Universal Robots PolyScope program: SandCube5.urp

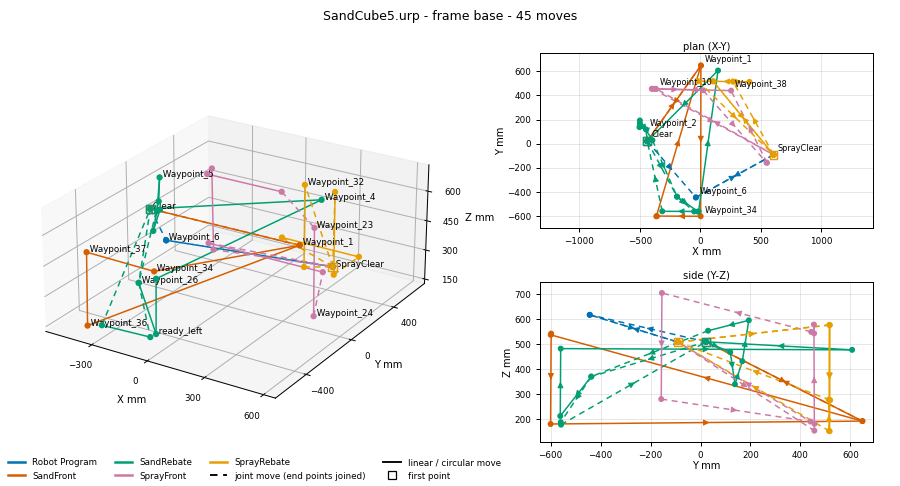
[picture p0: tool path of SandCube5.urp in frame base, 45 of 45 moves have a stored position in this frame; points joined in program order, loops and branches not executed]
Program SandCube5 (installation=sand5 directory=/programs createdIn=5.11.5.1010327 lastSavedIn=5.11.5.1010327 robotSerialNumber=20215500677)
Calibrated DH parameters: a=[0.000204, -0.239222, -0.391845, -0.000001, 0.000022, 0]; d=[0.162722, -355.808559, 353.37206, 2.570385, 0.099741, 0.099629]; alpha=[1.571124, 0.000988, 0.008295, 1.568963, -1.570303, 0]; deltaTheta=[0, -0.973091, 7.204745, 0.05153, 0, 0]
InitVariablesNode variables(variable(name=readyBackSand, expression=False), variable(name=readyFrontSand, expression=False), variable(name=readySpray, expression=False))
Robot Program (runOnlyOnce=false)
  Folder Main
    If readyFrontSand≟ True (checkContinuously=true)
      MoveJ speed 60 deg/s, acceleration 80 deg/s^2 (useActiveTCP=false positionType=JointAngles) tcp=DynabradeDual; feature=CubeFront
        Waypoint Clear: TCP in base x=-437.78 y=22.317 z=510.388 mm, rx=-1.2261 ry=-1.1914 rz=1.1915 rad; joints [-41.645, -103.017, 131.059, 99.527, -63.29, 31.09] deg; TCP offset x=3.18 y=114.64 z=98.2 mm, rx=-0.7854 ry=0 rz=0 rad; feature pose in base x=-591.611 y=-180.941 z=285.211 mm, rx=1.216 ry=1.1897 rz=1.1897 rad
        URCap Zero FT Sensor (Robotiq_Copilot, Robotiq Inc.) dataModel(NodeInitializedKey=true, WaitForSteadyWrenchOptionKey=true)
      Work := CubeFront
      Call SandFront
      Call SandRebate
      readyFrontSand := False
      Set DigitalOutput pin=digital_out[5]; digitalValue=0
    If readyBackSand≟ True (checkContinuously=true)
      Work := CubeFront
      Call SandFront
      readyBackSand := False
      Set DigitalOutput pin=digital_out[5]; digitalValue=0
    If readySpray≟ True (checkContinuously=true)
      MoveJ speed 60 deg/s, acceleration 80 deg/s^2 (useActiveTCP=false positionType=JointAngles) tcp=Spray; feature=SprayPlane
        Waypoint Waypoint_6: TCP in base x=-35.819 y=-443.732 z=618.465 mm, rx=1.57 ry=-0.053 rz=-0.0554 rad; joints [61.905, -86.892, 117.128, 101.277, -70.255, 21.732] deg; TCP offset x=20.839 y=-27.14 z=105.994 mm, rx=0.1226 ry=1.1769 rz=2.8697 rad; feature pose in base x=714.825 y=225.543 z=302.034 mm, rx=1.1969 ry=-1.2373 rz=-1.2135 rad
        Waypoint SprayClear: TCP in base x=607.137 y=-90.197 z=509.102 mm, rx=1.2034 ry=1.2067 rz=1.2159 rad; joints [154.541, -56.922, 94.352, -266.679, -69.476, 23.135] deg; TCP offset x=20.839 y=-27.14 z=105.994 mm, rx=0.1226 ry=1.1769 rz=2.8697 rad; feature pose in base x=807.673 y=110.818 z=310.566 mm, rx=1.2166 ry=-1.2106 rz=-1.2041 rad
        URCap Zero FT Sensor (Robotiq_Copilot, Robotiq Inc.) dataModel(NodeInitializedKey=true, WaitForSteadyWrenchOptionKey=true)
        Call SprayFront
        Call SprayRebate
        Waypoint Waypoint_6: TCP in base x=-35.819 y=-443.732 z=618.465 mm, rx=1.57 ry=-0.053 rz=-0.0554 rad; joints [61.905, -86.892, 117.128, 101.277, -70.255, 21.732] deg; TCP offset x=20.839 y=-27.14 z=105.994 mm, rx=0.1226 ry=1.1769 rz=2.8697 rad; feature pose in base x=714.825 y=225.543 z=302.034 mm, rx=1.1969 ry=-1.2373 rz=-1.2135 rad
        readySpray := False
  SuppressedNode
    Folder Chamfer
      MoveL speed 250 mm/s, acceleration 1200 mm/s^2 (useActiveTCP=true) feature=Base
        MoveJ speed 60 deg/s, acceleration 80 deg/s^2 (useActiveTCP=true) feature=CubeFront
          Waypoint Waypoint_14: TCP in base x=40.557 y=344.633 z=644.318 mm, rx=1.3155 ry=-1.3725 rz=-1.2523 rad; joints [213.145, -95.792, 65.461, -31.373, -65.462, -328.995] deg; TCP offset x=3.18 y=114.64 z=98.2 mm, rx=-0.7854 ry=0 rz=0 rad; feature pose in base x=6.058 y=653.089 z=192.929 mm, rx=1.5716 ry=0.003 rz=-0.0025 rad
          Waypoint Waypoint_15: TCP in base x=-6.602 y=417.802 z=666.352 mm, rx=-2.8064 ry=0.3635 rz=0.257 rad; joints [242.083, -106.85, 75.59, -118.753, -70.655, -356.384] deg
          Waypoint Waypoint_16: TCP in base x=7.321 y=653.157 z=552.583 mm, rx=-2.3553 ry=0.0014 rz=0.0042 rad; joints [252.243, -84.14, 86.654, -182.715, -72.191, -359.211] deg
        URCap Find Surface (Robotiq_Copilot, Robotiq Inc.) dataModel(NodeInitializedKey=true, ZeroSensorBeforeKey=true, WaitForSteadyWrenchOptionKey=false, ls_force=10.0, ls_distance=100.0, ls_speed=5.0, ls_if_distance=false, ls_if_force=false); state(isChildrenLocked=true)
          'Add Stop conditions from the Find Surface node'
        URCap Finishing Tool Control (Robotiq_Copilot, Robotiq Inc.) dataModel(ToolOutputNameKey=digital_out[0], HackTriggeringContributionIsDefinedMethodKey=true)
        Wait Sleep waitTime=0.5
        MoveDirectionNode (selectedDirection=XPlus toolParams=0.15, 1.2) feature(featureName=CubeFront)
          Until DISTANCE (allowActions=false deceleration=3 distanceNodeType=STOP) Distance=0.35; motionParameters(blendRadius=0)
        MoveDirectionNode (selectedDirection=ZMinus) feature=Joint_6_name
          Until DISTANCE (allowActions=false deceleration=3 distanceNodeType=STOP) Distance=0.025; motionParameters(blendRadius=0)
        URCap Finishing Tool Control (Robotiq_Copilot, Robotiq Inc.) dataModel(FinishingToolStateKey=false, ToolOutputNameKey=digital_out[0], HackTriggeringContributionIsDefinedMethodKey=true)
        Waypoint Waypoint_18: TCP in base x=366.179 y=605.982 z=520.828 mm, rx=-1.6861 ry=0.1385 rz=1.2496 rad; joints [208.374, -44.818, 51.064, -237.69, -37.068, -253.683] deg
        URCap Find Surface (Robotiq_Copilot, Robotiq Inc.) dataModel(NodeInitializedKey=true, ZeroSensorBeforeKey=true, WaitForSteadyWrenchOptionKey=false, ls_force=10.0, ls_distance=100.0, ls_speed=5.0, ls_if_distance=false, ls_if_force=false); state(isChildrenLocked=true)
          'Add Stop conditions from the Find Surface node'
        URCap Finishing Tool Control (Robotiq_Copilot, Robotiq Inc.) dataModel(ToolOutputNameKey=digital_out[0], HackTriggeringContributionIsDefinedMethodKey=true)
        MoveDirectionNode (selectedDirection=YMinus toolParams=0.15, 1.2) feature(featureName=CubeFront)
          Until DISTANCE (allowActions=false deceleration=3 distanceNodeType=STOP) Distance=0.35; motionParameters(blendRadius=0)
        URCap Finishing Tool Control (Robotiq_Copilot, Robotiq Inc.) dataModel(FinishingToolStateKey=false, ToolOutputNameKey=digital_out[0], HackTriggeringContributionIsDefinedMethodKey=true)
        MoveDirectionNode (selectedDirection=ZMinus) feature=Joint_6_name
          Until DISTANCE (allowActions=false deceleration=3 distanceNodeType=STOP) Distance=0.05; motionParameters(blendRadius=0)
        Waypoint Waypoint_20: TCP in base x=366.722 y=626.869 z=194.22 mm, rx=-1.1174 ry=-0.6786 rz=-0.9417 rad; joints [212.764, -30.352, 68.609, -330.279, -35.41, -327.866] deg
        URCap Find Surface (Robotiq_Copilot, Robotiq Inc.) dataModel(NodeInitializedKey=true, ZeroSensorBeforeKey=true, WaitForSteadyWrenchOptionKey=false, ls_force=10.0, ls_distance=100.0, ls_speed=5.0, ls_if_distance=false, ls_if_force=false); state(isChildrenLocked=true)
          'Add Stop conditions from the Find Surface node'
        URCap Finishing Tool Control (Robotiq_Copilot, Robotiq Inc.) dataModel(ToolOutputNameKey=digital_out[0], HackTriggeringContributionIsDefinedMethodKey=true)
        Waypoint Waypoint_19: motionParameters(jointSpeed=1.047198 jointAcceleration=1.396263 cartesianSpeed=0.05 cartesianAcceleration=1.2); TCP in base x=29.784 y=640.794 z=212.679 mm, rx=-1.2502 ry=-0.1072 rz=-0.0765 rad; joints [247.483, -34.268, 98.117, -310.948, -74.468, -342.493] deg
        URCap Finishing Tool Control (Robotiq_Copilot, Robotiq Inc.) dataModel(FinishingToolStateKey=false, ToolOutputNameKey=digital_out[0], HackTriggeringContributionIsDefinedMethodKey=true)
        MoveDirectionNode (selectedDirection=ZMinus) feature=Joint_6_name
          Until DISTANCE (allowActions=false deceleration=3 distanceNodeType=STOP) Distance=0.05; motionParameters(blendRadius=0)
Event  expression=digital_in[0]≠ True
  Set DigitalOutput pin=digital_out[0]; digitalValue=0
  Set DigitalOutput pin=digital_out[1]; digitalValue=0
  Halt
Event  expression=digital_in[1]≟ True
  readyFrontSand := True
  Set DigitalOutput pin=digital_out[5]; digitalValue=1
Event  expression=digital_in[2]≟ True
  readyBackSand := True
  Set DigitalOutput pin=digital_out[5]; digitalValue=1
Event  expression=digital_in[3]≟ True
  readySpray := True
SubProgram -> SandRebate
SubProgram -> SprayFront
SubProgram -> SprayRebate
SubProgram -> SandFront
SubProgram StartSpray [hidden by the author, left out]
SubProgram stopSpray [hidden by the author, left out]
SubProgram SandFront (keepSynchronizedWithDisk=false)
  Folder sandFront
    MoveJ speed 60 deg/s, acceleration 80 deg/s^2 (useActiveTCP=false positionType=JointAngles) tcp=DynabradeDual; feature=Work
      Waypoint Clear: TCP in base x=-437.78 y=22.317 z=510.388 mm, rx=-1.2261 ry=-1.1914 rz=1.1915 rad; joints [-41.645, -103.017, 131.059, 99.527, -63.29, 31.09] deg; TCP offset x=3.18 y=114.64 z=98.2 mm, rx=-0.7854 ry=0 rz=0 rad; feature pose in base x=-591.611 y=-180.941 z=285.211 mm, rx=1.216 ry=1.1897 rz=1.1897 rad
      SuppressedNode
        Waypoint Waypoint_35: TCP in base x=-544.551 y=45.618 z=509.072 mm, rx=-1.2092 ry=-1.2181 rz=1.2109 rad; joints [-31.988, -85.182, 115.602, 99.979, -68.031, 24.222] deg; TCP offset x=3.18 y=114.64 z=98.2 mm, rx=-0.7854 ry=0 rz=0 rad; feature pose in base x=-691.483 y=-161.421 z=282.725 mm, rx=1.203 ry=1.2097 rz=1.2171 rad
    MoveL speed 250 mm/s, acceleration 1200 mm/s^2 (useActiveTCP=false) tcp=DynabradeDual; feature=Work
      Waypoint Waypoint_1: TCP in base x=6.072 y=648.1 z=192.982 mm, rx=-1.5699 ry=0.0092 rz=0.0097 rad; joints [251.403, -67.593, 131.535, -110.394, 77.851, -166.352] deg; feature pose in base x=6.058 y=653.089 z=192.929 mm, rx=1.5716 ry=0.003 rz=-0.0025 rad
      URCap Zero FT Sensor (Robotiq_Copilot, Robotiq Inc.) dataModel(NodeInitializedKey=true, WaitForSteadyWrenchOptionKey=true)
      URCap Find Surface (Robotiq_Copilot, Robotiq Inc.) dataModel(NodeInitializedKey=true, WaitForSteadyWrenchOptionKey=false, ls_force=10.0, ls_distance=100.0, ls_speed=5.0, ZeroSensorBeforeKey=false, ls_if_distance=false, ls_if_force=false); state(isChildrenLocked=true)
        'Add Stop conditions from the Find Surface node'
      URCap Finishing Tool Control (Robotiq_Copilot, Robotiq Inc.) dataModel(ToolOutputNameKey=digital_out[0], HackTriggeringContributionIsDefinedMethodKey=true)
      Wait Sleep waitTime=0.5
    MoveL speed 60 mm/s, acceleration 1200 mm/s^2 (useActiveTCP=false) tcp=DynabradeDual; feature=Work
      Force Simple feature=Joint_6_name; selection=[0, 0, 1, 0, 0, 0]; wrench=[0, 0, 7, 0, 0, 0]; limitsForce=[0.15, 0.15, 0.15, 1.047198, 1.047198, 1.047198]; limitsMotion=[0.1, 0.1, 0.1, 0.349066, 0.349066, 0.349066]
        Waypoint Waypoint_34: TCP in base x=4.168 y=-599.662 z=538.228 mm, rx=0.1003 ry=-2.1628 rz=2.1762 rad; joints [69.8, -105.08, 109.114, -52.157, 72.617, -168.988] deg; feature pose in base x=2.048 y=-607.004 z=173.227 mm, rx=-0.0204 ry=-2.2235 rz=-2.2094 rad
        Waypoint Waypoint_37: TCP in base x=-357.721 y=-598.101 z=543.274 mm, rx=0.1002 ry=-2.1629 rz=2.1762 rad; joints [31.577, -86.57, 95.791, -75.508, 51.138, -132.637] deg
        Waypoint Waypoint_36: TCP in base x=-362.939 y=-600.337 z=181.342 mm, rx=0.1002 ry=-2.1628 rz=2.1761 rad; joints [31.404, -55.313, 118.507, -129.285, 51.013, -132.956] deg
        Waypoint Waypoint_1: TCP in base x=6.072 y=648.1 z=192.982 mm, rx=-1.5699 ry=0.0092 rz=0.0097 rad; joints [251.403, -67.593, 131.535, -110.394, 77.851, -166.352] deg; feature pose in base x=6.058 y=653.089 z=192.929 mm, rx=1.5716 ry=0.003 rz=-0.0025 rad
        URCap Finishing Tool Control (Robotiq_Copilot, Robotiq Inc.) dataModel(FinishingToolStateKey=false, ToolOutputNameKey=digital_out[0], HackTriggeringContributionIsDefinedMethodKey=true)
      MoveDirectionNode (selectedDirection=ZMinus) feature=Joint_6_name
        Until DISTANCE (allowActions=false deceleration=3 distanceNodeType=STOP) Distance=0.025; motionParameters(blendRadius=0)
    MoveJ speed 60 deg/s, acceleration 80 deg/s^2 (useActiveTCP=true positionType=JointAngles) feature=Work
      Waypoint Clear: TCP in base x=-437.78 y=22.317 z=510.388 mm, rx=-1.2261 ry=-1.1914 rz=1.1915 rad; joints [-41.645, -103.017, 131.059, 99.527, -63.29, 31.09] deg; TCP offset x=3.18 y=114.64 z=98.2 mm, rx=-0.7854 ry=0 rz=0 rad; feature pose in base x=-591.611 y=-180.941 z=285.211 mm, rx=1.216 ry=1.1897 rz=1.1897 rad
      SuppressedNode
        Waypoint Waypoint_35: TCP in base x=-544.551 y=45.618 z=509.072 mm, rx=-1.2092 ry=-1.2181 rz=1.2109 rad; joints [-31.988, -85.182, 115.602, 99.979, -68.031, 24.222] deg; TCP offset x=3.18 y=114.64 z=98.2 mm, rx=-0.7854 ry=0 rz=0 rad; feature pose in base x=-691.483 y=-161.421 z=282.725 mm, rx=1.203 ry=1.2097 rz=1.2171 rad
SubProgram SandRebate (keepSynchronizedWithDisk=false)
  Folder sandRebate
    MoveJ speed 60 deg/s, acceleration 80 deg/s^2 (useActiveTCP=false positionType=JointAngles) tcp=DynabradeDual; feature=CubeFront
      Waypoint Clear: TCP in base x=-437.78 y=22.317 z=510.388 mm, rx=-1.2261 ry=-1.1914 rz=1.1915 rad; joints [-41.645, -103.017, 131.059, 99.527, -63.29, 31.09] deg; TCP offset x=3.18 y=114.64 z=98.2 mm, rx=-0.7854 ry=0 rz=0 rad; feature pose in base x=-591.611 y=-180.941 z=285.211 mm, rx=1.216 ry=1.1897 rz=1.1897 rad
      MoveJ speed 60 deg/s, acceleration 80 deg/s^2 (useActiveTCP=false) tcp=DynabradeDual; feature=Work
        Waypoint Waypoint_26: TCP in base x=-191.756 y=-437.456 z=371.093 mm, rx=0.028 ry=2.2057 rz=-2.2199 rad; joints [21.356, -114.492, 145.455, -99.898, 50.061, -119.068] deg; TCP offset x=3.18 y=114.64 z=98.2 mm, rx=-0.7854 ry=0 rz=0 rad; feature pose in base x=2.048 y=-607.004 z=173.227 mm, rx=-0.0204 ry=-2.2235 rz=-2.2094 rad
      URCap Zero FT Sensor (Robotiq_Copilot, Robotiq Inc.) dataModel(NodeInitializedKey=true, WaitForSteadyWrenchOptionKey=true)
      MoveL speed 250 mm/s, acceleration 1200 mm/s^2 (useActiveTCP=false) tcp=DynabradeDual; feature=CubeFront
        Waypoint ready_left: TCP in base x=-17.184 y=-561.661 z=213.234 mm, rx=-0.6737 ry=1.48 rz=-0.6683 rad; joints [51.771, -52.432, 111.931, -157.066, 32.2, -30.92] deg
        URCap Find Surface (Robotiq_Copilot, Robotiq Inc.) dataModel(NodeInitializedKey=true, WaitForSteadyWrenchOptionKey=false, ls_force=10.0, ls_distance=100.0, ls_speed=5.0, ls_if_distance=false, ls_if_force=false, ZeroSensorBeforeKey=true); state(isChildrenLocked=true)
          'Add Stop conditions from the Find Surface node'
        URCap Finishing Tool Control (Robotiq_Copilot, Robotiq Inc.) dataModel(ToolOutputNameKey=digital_out[0], HackTriggeringContributionIsDefinedMethodKey=true)
        Wait Sleep waitTime=0.5
        Force Simple feature=Joint_6_name; selection=[0, 0, 1, 0, 0, 0]; wrench=[0, 0, 5, 0, 0, 0]; limitsForce=[0.15, 0.15, 0.15, 1.047198, 1.047198, 1.047198]; limitsMotion=[0.1, 0.1, 0.1, 0.349066, 0.349066, 0.349066]
          Waypoint Waypoint_44: motionParameters(jointSpeed=1.047198 jointAcceleration=1.396263 cartesianSpeed=0.05 cartesianAcceleration=1.2); TCP in base x=-13.375 y=-559.944 z=483.185 mm, rx=-1.5795 ry=0.9431 rz=-1.5593 rad; joints [55.751, -62.036, 88.983, -164.904, 66.281, -57.616] deg; TCP offset x=3.18 y=114.64 z=98.2 mm, rx=-0.7854 ry=0 rz=0 rad
        URCap Finishing Tool Control (Robotiq_Copilot, Robotiq Inc.) dataModel(ToolOutputNameKey=digital_out[0], HackTriggeringContributionIsDefinedMethodKey=true, FinishingToolStateKey=false)
        Waypoint Waypoint_4: TCP in base x=147.72 y=606.874 z=478.224 mm, rx=-0.8396 ry=-1.4025 rz=0.8394 rad; joints [229.161, -48.232, 67.407, -157.963, 71.791, -53.121] deg; TCP offset x=3.18 y=114.64 z=98.2 mm, rx=-0.7854 ry=0 rz=0 rad; feature pose in base x=85.344 y=655.608 z=190.328 mm, rx=1.5707 ry=0.001 rz=-0.0012 rad
        Waypoint Clear: TCP in base x=-437.78 y=22.317 z=510.388 mm, rx=-1.2261 ry=-1.1914 rz=1.1915 rad; joints [-41.645, -103.017, 131.059, 99.527, -63.29, 31.09] deg; TCP offset x=3.18 y=114.64 z=98.2 mm, rx=-0.7854 ry=0 rz=0 rad; feature pose in base x=-591.611 y=-180.941 z=285.211 mm, rx=1.216 ry=1.1897 rz=1.1897 rad
        Waypoint Waypoint_2: TCP in base x=-449.186 y=119.055 z=468.921 mm, rx=-1.5824 ry=0.0033 rz=-0.0189 rad; joints [355.989, -90.939, 116.285, -111.773, 135.96, -265.774] deg; TCP offset x=3.18 y=114.64 z=98.2 mm, rx=-0.7854 ry=0 rz=0 rad; feature pose in base x=-556.728 y=-197.219 z=289.992 mm, rx=1.1979 ry=1.1995 rz=1.1922 rad
        Waypoint Waypoint_3: TCP in base x=-502.582 y=137.86 z=340.388 mm, rx=-1.5824 ry=0.0034 rz=-0.0188 rad; joints [354.245, -73.54, 118.338, -129.583, 135.758, -263.461] deg; TCP offset x=3.18 y=114.64 z=98.2 mm, rx=-0.7854 ry=0 rz=0 rad
        URCap Find Surface (Robotiq_Copilot, Robotiq Inc.) dataModel(NodeInitializedKey=true, WaitForSteadyWrenchOptionKey=false, ls_force=10.0, ls_distance=100.0, ls_speed=5.0, ls_if_distance=false, ls_if_force=false, ZeroSensorBeforeKey=true); state(isChildrenLocked=true)
          'Add Stop conditions from the Find Surface node'
        URCap Finishing Tool Control (Robotiq_Copilot, Robotiq Inc.) dataModel(ToolOutputNameKey=digital_out[0], HackTriggeringContributionIsDefinedMethodKey=true)
        Wait Sleep waitTime=2
        Force Simple feature=Joint_6_name; selection=[0, 0, 1, 0, 0, 0]; wrench=[0, 0, 5, 0, 0, 0]; limitsForce=[0.15, 0.15, 0.15, 1.047198, 1.047198, 1.047198]; limitsMotion=[0.1, 0.1, 0.1, 0.349066, 0.349066, 0.349066]
          Waypoint Waypoint_8: motionParameters(jointSpeed=1.047198 jointAcceleration=1.396263 cartesianSpeed=0.1 cartesianAcceleration=1.2); TCP in base x=-499.275 y=167.355 z=432.595 mm, rx=-1.2269 ry=-1.1959 rz=-1.2362 rad; joints [-10.12, -84.222, 92.411, -7.899, 126.611, -269.865] deg; TCP offset x=3.18 y=114.64 z=98.2 mm, rx=-0.7854 ry=0 rz=0 rad; feature pose in base x=-558.85 y=-171.06 z=286.428 mm, rx=1.2201 ry=1.1846 rz=1.1887 rad
          Waypoint Waypoint_5: motionParameters(jointSpeed=1.047198 jointAcceleration=1.396263 cartesianSpeed=0.05 cartesianAcceleration=1.2); TCP in base x=-499.119 y=193.296 z=596.509 mm, rx=-1.074 ry=-1.4158 rz=-1.4514 rad; joints [-13.477, -78.664, 59.577, 33.743, 123.4, -274.104] deg; TCP offset x=3.18 y=114.64 z=98.2 mm, rx=-0.7854 ry=0 rz=0 rad
          MoveDirectionNode (selectedDirection=ZMinus) feature=Joint_6_name
            Until DISTANCE (allowActions=false deceleration=3 distanceNodeType=STOP) Distance=0.05; motionParameters(blendRadius=0)
        URCap Finishing Tool Control (Robotiq_Copilot, Robotiq Inc.) dataModel(FinishingToolStateKey=false, ToolOutputNameKey=digital_out[0], HackTriggeringContributionIsDefinedMethodKey=true)
        Waypoint Waypoint_17: TCP in base x=-395.175 y=30.149 z=554.775 mm, rx=-1.1505 ry=-1.3153 rz=-1.1331 rad; joints [8.831, -95.06, 83.539, 16.597, 137.575, -265.28] deg; TCP offset x=3.18 y=114.64 z=98.2 mm, rx=-0.7854 ry=0 rz=0 rad; feature pose in base x=-581.609 y=-292.901 z=304.023 mm, rx=1.2041 ry=1.185 rz=1.1651 rad
        MoveJ speed 60 deg/s, acceleration 80 deg/s^2 (useActiveTCP=false) tcp=DynabradeDual; feature=Work
          Waypoint Waypoint_26: TCP in base x=-191.756 y=-437.456 z=371.093 mm, rx=0.028 ry=2.2057 rz=-2.2199 rad; joints [21.356, -114.492, 145.455, -99.898, 50.061, -119.068] deg; feature pose in base x=2.048 y=-607.004 z=173.227 mm, rx=-0.0204 ry=-2.2235 rz=-2.2094 rad
        MoveJ speed 60 deg/s, acceleration 80 deg/s^2 (useActiveTCP=false) tcp=DynabradeDual; feature=CubeFront
          Waypoint Waypoint_31: TCP in base x=-50.065 y=-559.682 z=188.667 mm, rx=2.5929 ry=-1.748 rz=-0.0179 rad; joints [66.855, -74.84, 90.337, -71.013, -60.355, -144.5] deg; TCP offset x=3.18 y=114.64 z=98.2 mm, rx=-0.7854 ry=0 rz=0 rad
          URCap Zero FT Sensor (Robotiq_Copilot, Robotiq Inc.) dataModel(NodeInitializedKey=true, WaitForSteadyWrenchOptionKey=true)
        URCap Find Surface (Robotiq_Copilot, Robotiq Inc.) dataModel(NodeInitializedKey=true, ZeroSensorBeforeKey=true, WaitForSteadyWrenchOptionKey=false, ls_force=10.0, ls_distance=100.0, ls_speed=5.0, ls_if_distance=false, ls_if_force=false); state(isChildrenLocked=true)
          'Add Stop conditions from the Find Surface node'
        URCap Finishing Tool Control (Robotiq_Copilot, Robotiq Inc.) dataModel(ToolOutputNameKey=digital_out[0], HackTriggeringContributionIsDefinedMethodKey=true)
        Wait Sleep waitTime=0.5
        Force Frame feature=Joint_6_name; selection=[0, 0, 1, 0, 0, 0]; wrench=[0, 0, 5, 0, 0, 0]; limitsForce=[0.15, 0.15, 0.15, 1.047198, 1.047198, 1.047198]; limitsMotion=[0.1, 0.1, 0.1, 0.349066, 0.349066, 0.349066]
          Waypoint Waypoint_7: motionParameters(jointSpeed=1.047198 jointAcceleration=1.396263 cartesianSpeed=0.05 cartesianAcceleration=1.2); TCP in base x=-313.929 y=-558.619 z=178.607 mm, rx=1.8205 ry=-2.5415 rz=-0.0103 rad; joints [43.867, -66.795, 83.357, -82.807, -51.116, -125.979] deg; TCP offset x=3.18 y=114.64 z=98.2 mm, rx=-0.7854 ry=0 rz=0 rad
        URCap Finishing Tool Control (Robotiq_Copilot, Robotiq Inc.) dataModel(FinishingToolStateKey=false, ToolOutputNameKey=digital_out[0], HackTriggeringContributionIsDefinedMethodKey=true)
        MoveDirectionNode (selectedDirection=ZPlus)
          Until DISTANCE (allowActions=false deceleration=3 distanceNodeType=STOP) Distance=0.05; motionParameters(blendRadius=0)
        SuppressedNode
          Waypoint Waypoint_13: TCP in base x=343.245 y=349.195 z=234.967 mm, rx=-1.8514 ry=-2.5381 rz=0.0001 rad; joints [208.052, -81.166, 89.339, -53.576, -82.434, -172.912] deg; TCP offset x=3.18 y=114.64 z=98.2 mm, rx=-0.7854 ry=0 rz=0 rad; feature pose in base x=9.685 y=618.378 z=176.869 mm, rx=1.5687 ry=-0.014 rz=-0.0074 rad
        SuppressedNode
          Waypoint Waypoint_9: TCP in base x=-0.811 y=492.962 z=588.061 mm, rx=-1.9827 ry=-0.1778 rz=-0.0774 rad; joints [237.765, -113.533, 89.133, -2.101, 52.621, -171.272] deg
      Waypoint Clear: TCP in base x=-437.78 y=22.317 z=510.388 mm, rx=-1.2261 ry=-1.1914 rz=1.1915 rad; joints [-41.645, -103.017, 131.059, 99.527, -63.29, 31.09] deg; TCP offset x=3.18 y=114.64 z=98.2 mm, rx=-0.7854 ry=0 rz=0 rad; feature pose in base x=-591.611 y=-180.941 z=285.211 mm, rx=1.216 ry=1.1897 rz=1.1897 rad
SubProgram SprayFront (keepSynchronizedWithDisk=false)
  Folder SprayFront
    MoveJ speed 60 deg/s, acceleration 80 deg/s^2 (useActiveTCP=false) tcp=Spray; feature=SprayPlane
      Waypoint SprayClear: TCP in base x=607.137 y=-90.197 z=509.102 mm, rx=1.2034 ry=1.2067 rz=1.2159 rad; joints [154.541, -56.922, 94.352, -266.679, -69.476, 23.135] deg; TCP offset x=20.839 y=-27.14 z=105.994 mm, rx=0.1226 ry=1.1769 rz=2.8697 rad; feature pose in base x=807.673 y=110.818 z=310.566 mm, rx=1.2166 ry=-1.2106 rz=-1.2041 rad
    MoveJ speed 60 deg/s, acceleration 80 deg/s^2 (useActiveTCP=false) tcp=Spray; feature=SprayPlane
      Waypoint Waypoint_10: TCP in base x=-366.88 y=455.74 z=154.683 mm, rx=-1.1923 ry=1.2085 rz=1.1804 rad; joints [282.195, -40.36, 126.156, -261.512, -59.605, -89.075] deg; TCP offset x=20.839 y=-27.14 z=105.994 mm, rx=0.1226 ry=1.1769 rz=2.8697 rad; feature pose in base x=-366.784 y=580.679 z=180.17 mm, rx=1.5749 ry=-0.0329 rz=-0.0106 rad
      Set DigitalOutput pin=digital_out[4]; digitalValue=1
    MoveL speed 100 mm/s, acceleration 1200 mm/s^2 (useActiveTCP=true) feature=SprayPlane
      Waypoint Waypoint_12: TCP in base x=-372.961 y=453.99 z=579.608 mm, rx=-1.1924 ry=1.2084 rz=1.1805 rad; joints [283.1, -92.847, 109.867, -192.963, -60.146, -88.612] deg
      Set DigitalOutput pin=digital_out[4]; digitalValue=0
      MoveDirectionNode (selectedDirection=ZMinus toolParams=0.2, 1.2) feature=Joint_6_name
        Until DISTANCE (allowActions=false deceleration=3 distanceNodeType=STOP) Distance=0.1; motionParameters(blendRadius=0)
    MoveJ speed 60 deg/s, acceleration 80 deg/s^2 (useActiveTCP=false) tcp=Spray; feature=SprayPlane
      Waypoint Waypoint_21: TCP in base x=-400.443 y=454.966 z=544.225 mm, rx=-1.5663 ry=0.0105 rz=-0.0329 rad; joints [305.438, -86.323, 77.292, -117.871, -118.512, -147.771] deg
      Set DigitalOutput pin=digital_out[4]; digitalValue=1
    MoveL speed 100 mm/s, acceleration 1200 mm/s^2 (useActiveTCP=false) tcp=Spray; feature=SprayPlane
      Waypoint Waypoint_22: TCP in base x=24.363 y=443.181 z=550.193 mm, rx=-1.5664 ry=0.0106 rz=-0.0328 rad; joints [239.529, -113.419, 99.688, -119.587, -73.088, -197.229] deg
      Set DigitalOutput pin=digital_out[4]; digitalValue=0
      MoveDirectionNode (selectedDirection=ZMinus toolParams=0.2, 1.2) feature=Joint_6_name
        Until DISTANCE (allowActions=false deceleration=3 distanceNodeType=STOP) Distance=0.1; motionParameters(blendRadius=0)
    MoveJ speed 60 deg/s, acceleration 80 deg/s^2 (useActiveTCP=false) tcp=Spray; feature=SprayPlane
      Waypoint Waypoint_23: TCP in base x=548.641 y=-154.61 z=706.095 mm, rx=-0.0121 ry=1.5616 rz=0.002 rad; joints [128.296, -68.562, 32.652, 13.403, -7.79, -244.639] deg; TCP offset x=20.839 y=-27.14 z=105.994 mm, rx=0.1226 ry=1.1769 rz=2.8697 rad; feature pose in base x=674.096 y=208.92 z=304.834 mm, rx=1.2154 ry=-1.2124 rz=-1.1935 rad
      Set DigitalOutput pin=digital_out[4]; digitalValue=1
    MoveL speed 100 mm/s, acceleration 1200 mm/s^2 (useActiveTCP=false) tcp=Spray; feature=SprayPlane
      Waypoint Waypoint_24: TCP in base x=552.545 y=-157.368 z=281.062 mm, rx=-0.0121 ry=1.5615 rz=0.0019 rad; joints [128.403, -70.766, 101.674, -54.987, -7.187, -243.057] deg
      Set DigitalOutput pin=digital_out[4]; digitalValue=0
      MoveDirectionNode (selectedDirection=ZMinus toolParams=0.2, 1.2) feature=Joint_6_name
        Until DISTANCE (allowActions=false deceleration=3 distanceNodeType=STOP) Distance=0.1; motionParameters(blendRadius=0)
      MoveDirectionNode (selectedDirection=ZPlus) feature=Base
        Until DISTANCE (allowActions=false deceleration=3 distanceNodeType=STOP) Distance=0.1; motionParameters(blendRadius=0)
    MoveJ speed 60 deg/s, acceleration 80 deg/s^2 (useActiveTCP=false) tcp=Spray; feature=SprayPlane
      Waypoint Waypoint_38: TCP in base x=255.883 y=440.293 z=191.235 mm, rx=-1.5741 ry=0.008 rz=-0.0287 rad; joints [210.744, -86.11, 132.363, -168.194, -55.616, -222.536] deg; TCP offset x=20.839 y=-27.14 z=105.994 mm, rx=0.1226 ry=1.1769 rz=2.8697 rad; feature pose in base x=-141.025 y=574.651 z=182.515 mm, rx=1.5672 ry=-0.0288 rz=-0.0081 rad
      Set DigitalOutput pin=digital_out[4]; digitalValue=1
    MoveL speed 100 mm/s, acceleration 1200 mm/s^2 (useActiveTCP=false) tcp=Spray; feature=SprayPlane
      Waypoint Waypoint_25: TCP in base x=-395.272 y=456.409 z=182.261 mm, rx=-1.5664 ry=0.0105 rz=-0.0328 rad; joints [304.782, -71.234, 116.575, -172.386, -118.444, -148.069] deg; TCP offset x=20.839 y=-27.14 z=105.994 mm, rx=0.1226 ry=1.1769 rz=2.8697 rad; feature pose in base x=-366.784 y=580.679 z=180.17 mm, rx=1.5749 ry=-0.0329 rz=-0.0106 rad
      Set DigitalOutput pin=digital_out[4]; digitalValue=0
      MoveDirectionNode (selectedDirection=ZMinus toolParams=0.2, 1.2) feature=Joint_6_name
        Until DISTANCE (allowActions=false deceleration=3 distanceNodeType=STOP) Distance=0.1; motionParameters(blendRadius=0)
    MoveJ speed 60 deg/s, acceleration 80 deg/s^2 (useActiveTCP=false) tcp=Spray; feature=SprayPlane
      Waypoint SprayClear: TCP in base x=607.137 y=-90.197 z=509.102 mm, rx=1.2034 ry=1.2067 rz=1.2159 rad; joints [154.541, -56.922, 94.352, -266.679, -69.476, 23.135] deg; TCP offset x=20.839 y=-27.14 z=105.994 mm, rx=0.1226 ry=1.1769 rz=2.8697 rad; feature pose in base x=807.673 y=110.818 z=310.566 mm, rx=1.2166 ry=-1.2106 rz=-1.2041 rad
SubProgram SprayRebate (keepSynchronizedWithDisk=false)
  Folder SprayRebate
    MoveJ speed 60 deg/s, acceleration 80 deg/s^2 (useActiveTCP=false) tcp=Spray; feature=SprayPlane
      Waypoint SprayClear: TCP in base x=607.137 y=-90.197 z=509.102 mm, rx=1.2034 ry=1.2067 rz=1.2159 rad; joints [154.541, -56.922, 94.352, -266.679, -69.476, 23.135] deg
    MoveJ speed 60 deg/s, acceleration 80 deg/s^2 (useActiveTCP=false) tcp=Spray; feature=SprayPlane
      Waypoint Waypoint_28: TCP in base x=271.667 y=515.614 z=578.139 mm, rx=-0.606 ry=1.4822 rz=0.6004 rad; joints [208.011, -87.406, 104.797, -191.165, -29.317, -91.698] deg; feature pose in base x=9.685 y=618.378 z=176.869 mm, rx=1.5687 ry=-0.014 rz=-0.0074 rad
      Set DigitalOutput pin=digital_out[4]; digitalValue=1
    MoveL speed 100 mm/s, acceleration 1200 mm/s^2 (useActiveTCP=false) tcp=Spray; feature=SprayPlane
      Waypoint Waypoint_27: TCP in base x=273.408 y=514.734 z=153.162 mm, rx=-0.606 ry=1.4823 rz=0.6004 rad; joints [207.859, -39.21, 119.689, -253.722, -29.522, -92.302] deg
      Set DigitalOutput pin=digital_out[4]; digitalValue=0
      MoveDirectionNode (selectedDirection=ZMinus toolParams=0.2, 1.2) feature(featureName=CubeFront)
        Until DISTANCE (allowActions=false deceleration=3 distanceNodeType=STOP) Distance=0.2; motionParameters(blendRadius=0)
    MoveJ speed 60 deg/s, acceleration 80 deg/s^2 (useActiveTCP=false) tcp=Spray; feature=SprayPlane
      Waypoint Waypoint_29: TCP in base x=407.829 y=513.19 z=278.745 mm, rx=0.0171 ry=2.8953 rz=1.196 rad; joints [202.265, -49.904, 107.859, -237.705, -20.006, 3.393] deg; TCP offset x=20.839 y=-27.14 z=105.994 mm, rx=0.1226 ry=1.1769 rz=2.8697 rad
      Set DigitalOutput pin=digital_out[4]; digitalValue=1
    MoveL speed 100 mm/s, acceleration 1200 mm/s^2 (useActiveTCP=false) tcp=Spray; feature=SprayPlane
      Waypoint Waypoint_30: TCP in base x=-17.094 y=518.98 z=276.97 mm, rx=0.0171 ry=2.8954 rz=1.196 rad; joints [250.228, -61.644, 139.534, -257.5, -68.041, 3.56] deg; TCP offset x=20.839 y=-27.14 z=105.994 mm, rx=0.1226 ry=1.1769 rz=2.8697 rad
      Set DigitalOutput pin=digital_out[4]; digitalValue=0
      MoveDirectionNode (selectedDirection=ZMinus toolParams=0.2, 1.2) feature(featureName=CubeFront)
        Until DISTANCE (allowActions=false deceleration=3 distanceNodeType=STOP) Distance=0.2; motionParameters(blendRadius=0)
    MoveJ speed 60 deg/s, acceleration 80 deg/s^2 (useActiveTCP=false) tcp=Spray; feature=SprayPlane
      Waypoint SprayClear: TCP in base x=607.137 y=-90.197 z=509.102 mm, rx=1.2034 ry=1.2067 rz=1.2159 rad; joints [154.541, -56.922, 94.352, -266.679, -69.476, 23.135] deg; feature pose in base x=807.673 y=110.818 z=310.566 mm, rx=1.2166 ry=-1.2106 rz=-1.2041 rad
    MoveL speed 100 mm/s, acceleration 1200 mm/s^2 (useActiveTCP=false) tcp=Spray; feature=SprayPlane
      MoveDirectionNode (selectedDirection=ZMinus toolParams=0.2, 1.2) feature(featureName=CubeFront)
        Until DISTANCE (allowActions=false deceleration=3 distanceNodeType=STOP) Distance=0.1; motionParameters(blendRadius=0)
    MoveJ speed 60 deg/s, acceleration 80 deg/s^2 (useActiveTCP=false) tcp=Spray; feature=SprayPlane
      Waypoint Waypoint_32: TCP in base x=106.648 y=517.867 z=577.433 mm, rx=-0.6252 ry=-1.4837 rz=-0.6245 rad; joints [231.305, -102.456, 86.054, 11.982, 51.705, -83.541] deg; feature pose in base x=9.685 y=618.378 z=176.869 mm, rx=1.5687 ry=-0.014 rz=-0.0074 rad
      Set DigitalOutput pin=digital_out[4]; digitalValue=1
    MoveL speed 100 mm/s, acceleration 1200 mm/s^2 (useActiveTCP=false) tcp=Spray; feature=SprayPlane
      Waypoint Waypoint_33: TCP in base x=108.397 y=516.974 z=152.506 mm, rx=-0.6252 ry=-1.4837 rz=-0.6245 rad; joints [230.83, -82.04, 136.774, -59.04, 51.734, -83.726] deg
      Set DigitalOutput pin=digital_out[4]; digitalValue=0
      MoveDirectionNode (selectedDirection=ZMinus toolParams=0.2, 1.2) feature(featureName=CubeFront)
        Until DISTANCE (allowActions=false deceleration=3 distanceNodeType=STOP) Distance=0.2; motionParameters(blendRadius=0)
    MoveJ speed 60 deg/s, acceleration 80 deg/s^2 (useActiveTCP=false) tcp=Spray; feature=SprayPlane
      Waypoint SprayClear: TCP in base x=607.137 y=-90.197 z=509.102 mm, rx=1.2034 ry=1.2067 rz=1.2159 rad; joints [154.541, -56.922, 94.352, -266.679, -69.476, 23.135] deg; feature pose in base x=807.673 y=110.818 z=310.566 mm, rx=1.2166 ry=-1.2106 rz=-1.2041 rad
